PROGRAM MAIN
VAR
	fbBottle : FB_BottleFiller;
	bFlag : BOOL := TRUE;
	nNum : INT := 43;
END_VAR

fbBottle.StartFilling();

END_PROGRAM

(* stored: Version 1.1.0.1, ProductVersion 3.1.4024.16
   POU MAIN: Id {31fe5ed8-789a-43d7-9bb7-c38f88336644}, SpecialFunc None *)
